Yaskawa INFORM job: WELDING-CMF100-ST2-FRONT.JBI

/JOB
//NAME WELDING-CMF100-ST2-FRONT
//POS
///NPOS 16,16,16,1,0,0
///TOOL 0
///POSTYPE PULSE
///PULSE
C00000=164669,-36340,-21106,52796,46739,16769
C00001=179001,-11276,-30769,96775,50105,-10318
C00002=170456,7256,-18069,103183,54177,-15188
C00003=171136,34534,-45795,140489,9656,-36018
C00004=171136,34289,-45736,140475,9803,-35976
C00005=171051,33990,-46063,140532,9761,-36011
C00006=169630,9662,-17399,105842,54041,-16481
C00007=169582,9756,-17356,105905,54060,-16516
C00008=169591,9722,-17474,105990,54028,-16574
C00009=169638,9630,-17519,105931,54009,-16541
C00010=139580,49357,71591,2475,27844,42830
C00011=139461,52784,76778,2212,25401,42897
C00012=142088,15246,34290,8811,48294,40874
C00013=141949,-14096,-14463,46727,74302,20109
C00014=126786,-51503,-34655,-20249,70608,58781
C00015=111202,-18113,-15031,-8392,50715,49810
BC00000=294004
BC00001=324712
BC00002=324712
BC00003=324712
BC00004=324712
BC00005=324712
BC00006=324712
BC00007=324712
BC00008=324712
BC00009=324712
BC00010=271716
BC00011=271716
BC00012=271716
BC00013=271716
BC00014=271716
BC00015=274290
EC00000=2040560
EC00001=2040560
EC00002=2040560
EC00003=2402229
EC00004=2402229
EC00005=2402229
EC00006=2049475
EC00007=1030579
EC00008=1834
EC00009=-988925
EC00010=-1528017
EC00011=-1528017
EC00012=-1047896
EC00013=-1047896
EC00014=-1047896
EC00015=-1022546
///USER 10
///POSTYPE USER
///RECTAN
///RCONF 0,0,0,0,0,0,0,0,0,0,0,0,0,0,0,0,0,0,0,0,0,0,0,0
P00049=2.600,0.000,0.000,0.0000,0.0000,0.0000
//INST
///DATE 2018/10/02 11:04
///ATTR SC,RW
///GROUP1 RB1,BS1
///GROUP2 ST2
NOP
'***** welding station 1 front
MOVJ C00000 BC00000 VJ=25.00  +MOVJ EC00000 VJ=100.00
'***** go to start pos
SMOVL C00001 BC00001 V=166.7 PL=0  +MOVJ EC00001
SFTON P049 UF#(20)
SMOVL C00002 BC00002 V=83.3  +MOVJ EC00002
SMOVC C00003 BC00003 V=83.3 PL=0  +MOVJ EC00003  //start welding
DOUT OT#(656) OFF
TIMER T=0.50
DOUT OT#(656) ON
MACRO1 MJ#(5) ARGF2
SREFP 1 C00004 BC00004  +REFP EC00004
SREFP 2 C00005 BC00005  +REFP EC00005
ARCON ASF#(1)
SWVON WEV#(1)
SMOVC C00006 BC00006 V=I000  +MOVJ EC00006
SMOVC C00007 BC00007 V=I000  +MOVJ EC00007
SMOVC C00008 BC00008 V=I000  +MOVJ EC00008
SMOVC C00009 BC00009 V=I000  +MOVJ EC00009
SMOVC C00010 BC00010 V=I000  +MOVJ EC00010
SMOVC C00011 BC00011 V=I000  +MOVJ EC00011
ARCOF
SMOVL C00012 BC00012 V=I000  +MOVJ EC00012
MACRO1 MJ#(5) ARGF5
DOUT OT#(656) OFF
SWVOF
TIMER T=5.00
'***** go to end position
SMOVL C00013 BC00013 V=83.3 PL=0  +MOVJ EC00013
SMOVL C00014 BC00014 V=83.3  +MOVJ EC00014
MOVL C00015 BC00015 V=166.7  +MOVJ EC00015 VJ=100.00
SFTOF
END
